TYPE ServicesStatuses :
STRUCT
	initializationStatus: InitializationStatus;
	healthStatus: HealthStatus;
	busyStatus: BusyStatus;
	operatingStatus: OperatingStatus;
END_STRUCT
END_TYPE

(* stored: Version 1.1.0.1, ProductVersion 3.1.4019.2
   DUT ServicesStatuses: Id {e574acf7-8a6e-4a96-b2dc-de20129681ea} *)
